ABB RobotStudio station: conveyor.rsstn

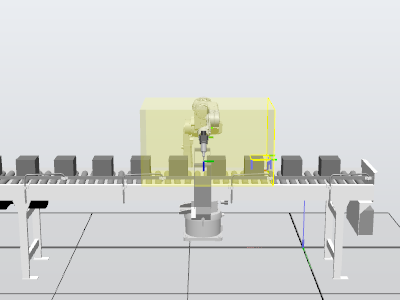
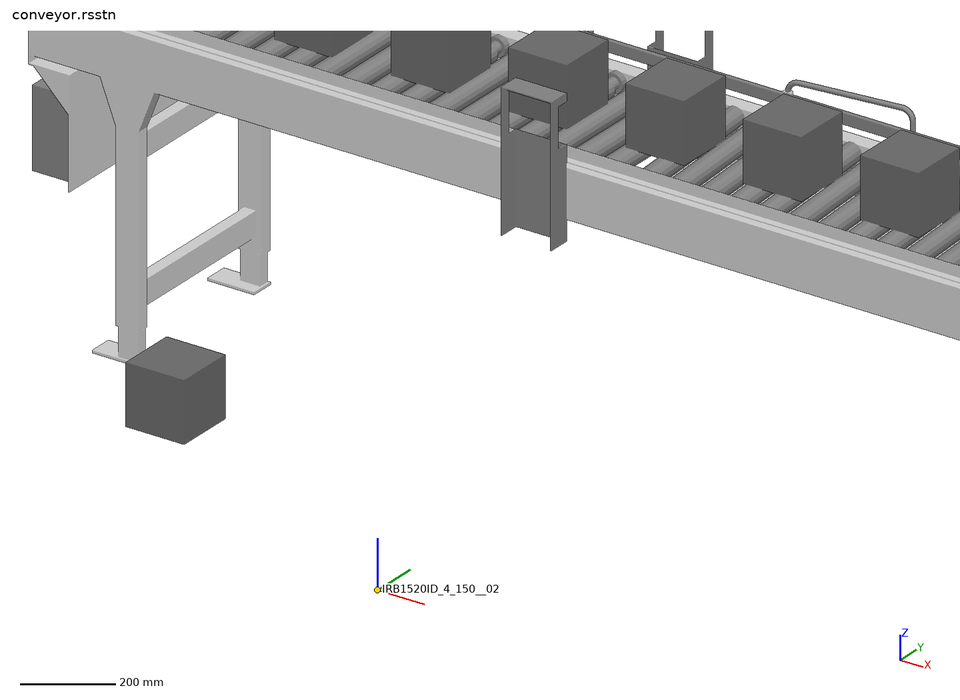
[picture v1: parts stored in the station drawn from their meshes, with robot base, taught points and paths (robot models come from the ABB library and are not in the file)]
Station Station (saved by RobotStudio 22.3.10141.1)
Controller Controller22, task T_ROB1: task frame (RAPID world) sits at (353.54, 291.96, 775) mm in the station
Controller Controller22
  mechanical unit ROB_1: IRB1520ID_4_150__02, 6 joints, base frame (527.64, -629.92, -775) mm, rotated rx 0 ry 0 rz 90 deg
  mechanical unit CNV1: ?, 1 joints, base frame (0, 0, 0) mm
Layout (positions relative to the parent item):
  - IRB1520ID_4_150__02 [mechanism, from Robots\IRB1520ID_4_150_G_02.rslib] at (881.18, -337.95, 0) mm, rotated rx 0 ry 0 rz 90 deg; joint values [0, 0, 0, 0, 0.5236, 0] (rad or m)
  - MyTool [mechanism, from Training Objects\myTool.rslib] at (881.18, 718.25, 1143) mm, rotated rx 180 ry 60 rz -90 deg
  - Conveyor [conveyor]
    - 400_guide [part] at (-421.3, 289.46, 0) mm, size 3033 x 590 x 945 mm
    - box [part], size 150 x 150 x 150 mm
    - ConveyorObject_358 [conveyorobject] at (2504.74, 291.96, 775) mm
      - box [part] at (0, 100, 0) mm, size 150 x 150 x 150 mm
    - ConveyorObject_359 [conveyorobject] at (2204.74, 291.96, 775) mm
      - box [part] at (0, 100, 0) mm, size 150 x 150 x 150 mm
    - ConveyorObject_360 [conveyorobject] at (1904.74, 291.96, 775) mm
      - box [part] at (0, 100, 0) mm, size 150 x 150 x 150 mm
    - ConveyorObject_361 [conveyorobject] at (1604.74, 291.96, 775) mm
      - box [part] at (0, 100, 0) mm, size 150 x 150 x 150 mm
    - ConveyorObject_362 [conveyorobject] at (1304.74, 291.96, 775) mm
      - box [part] at (0, 100, 0) mm, size 150 x 150 x 150 mm
    - ConveyorObject_363 [conveyorobject] at (1004.74, 291.96, 775) mm
      - box [part] at (0, 100, 0) mm, size 150 x 150 x 150 mm
    - ConveyorObject_364 [conveyorobject] at (704.74, 291.96, 775) mm
      - box [part] at (0, 100, 0) mm, size 150 x 150 x 150 mm
    - ConveyorObject_365 [conveyorobject] at (404.74, 291.96, 775) mm
      - box [part] at (0, 100, 0) mm, size 150 x 150 x 150 mm
    - ConveyorObject_366 [conveyorobject] at (104.74, 291.96, 775) mm
      - box [part] at (0, 100, 0) mm, size 150 x 150 x 150 mm
    - ConveyorObject_367 [conveyorobject] at (-195.26, 291.96, 775) mm
      - box [part] at (0, 100, 0) mm, size 150 x 150 x 150 mm
Attachment: MyTool is attached to IRB1520ID_4_150__02 / Link6
Conveyor tracking Connection: unit CNV1, TravelOffset=0.7, QueueTrackDistance=0, StartWindowWidth=1, SyncSeparation=0.1, CountsPerMeter=10000
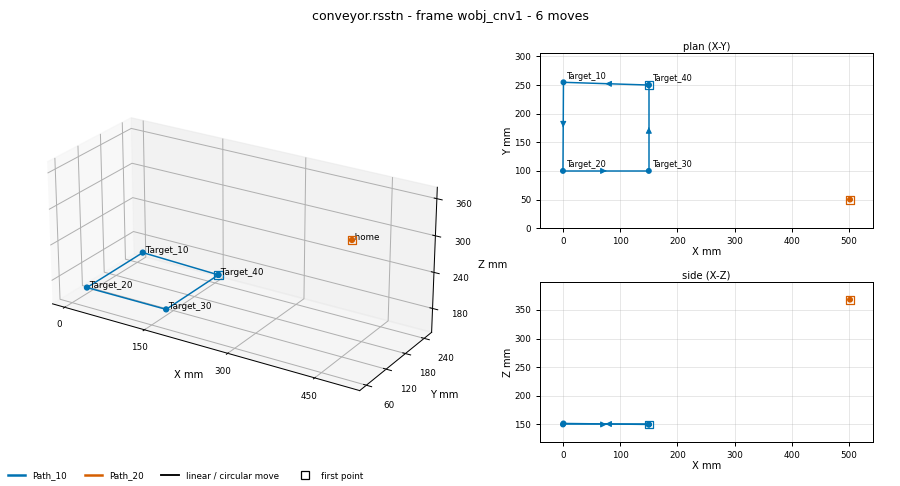
[picture p0: tool path of conveyor.rsstn in frame wobj_cnv1, 6 of 6 moves have a stored position in this frame; points joined in program order, loops and branches not executed]
Targets, tools, work objects and paths stored in the station, written as RAPID:
! task T_ROB1
MODULE CalibData
  TASK PERS wobjdata wobj_cnv1:=[FALSE,FALSE,"CNV1",[[0,0,0],[1,0,0,0]],[[0,0,0],[1,0,0,0]]];
  PERS tooldata MyTool:=[TRUE,[[31.792631019,0,229.638935148],[0.945518576,0,0.325568154,0]],[1,[0,0,1],[1,0,0,0],0,0,0]];
ENDMODULE

! task T_ROB1
MODULE Module1
  CONST robtarget home:=[[501.522589301,49.908702126,368.000030749],[0.353553395,-0.612372433,0.612372433,0.353553395],[0,-1,0,0],[9E+09,9E+09,9E+09,9E+09,9E+09,0]];
  CONST robtarget Target_10:=[[0.863881796,254.78672145,151.764208865],[0.134922335,-0.694115254,0.694115232,0.134922285],[0,1,-2,1],[9E+09,9E+09,9E+09,9E+09,9E+09,0]];
  CONST robtarget Target_20:=[[-0.000020312,100.000008756,149.999988617],[0.134922306,-0.694115256,0.694115241,0.134922254],[0,1,-2,1],[9E+09,9E+09,9E+09,9E+09,9E+09,0]];
  CONST robtarget Target_30:=[[150.000021683,100.000042154,149.999993709],[0.134922337,-0.69411529,0.694115223,0.134922147],[0,1,-2,1],[9E+09,9E+09,9E+09,9E+09,9E+09,0]];
  CONST robtarget Target_40:=[[149.999946962,250.000040029,149.999986787],[0.134922265,-0.694115287,0.694115236,0.134922162],[0,1,-2,1],[9E+09,9E+09,9E+09,9E+09,9E+09,0]];
  PROC Path_10()
    MoveL Target_40,v1000,fine,MyTool\WObj:=wobj_cnv1;
    MoveL Target_10,v1000,fine,MyTool\WObj:=wobj_cnv1;
    MoveL Target_20,v1000,fine,MyTool\WObj:=wobj_cnv1;
    MoveL Target_30,v1000,fine,MyTool\WObj:=wobj_cnv1;
    MoveL Target_40,v1000,fine,MyTool\WObj:=wobj_cnv1;
  ENDPROC
  PROC Path_20()
    MoveL home,v1000,z100,MyTool\WObj:=wobj_cnv1;
    ActUnit CNV1;
    WaitWObj wobj_cnv1;
    Path_10;
    WaitWObj wobj_cnv1;
  ENDPROC
ENDMODULE

